// TIA Portal V16 export
// export: Created 2021-11-12T13:32:20.8858342Z, ExportSetting WithDefaults, DisplayName Totally Integrated Automation Portal, DisplayVersion V16 Update 3, DisplayName TIA Portal Version Control Interface, DisplayVersion V16 Update 2, DisplayName TIA Portal Openness, DisplayVersion V16 Update 3, DisplayName SINAMICS Startdrive Advanced, DisplayVersion V16 Update 5, DisplayName SINAMICS Startdrive G130, G150, S120, S150, SINAMICS MV, S210, DisplayVersion V16 Update 5, DisplayName SINAMICS Startdrive G110M, G120, G120C, G120D, G120P, G115D, DisplayVersion V16 Update 5, DisplayName STEP 7 Professional, DisplayVersion V16 Update 3, DisplayName STEP 7 Safety, DisplayVersion V16, DisplayName WinCC UA Professional, DisplayVersion V16 Update 3
DATA_BLOCK "HMI_PARAM_1R5"   // DB91
{ S7_Optimized_Access := 'TRUE' }
VERSION : 0.1
// stored: AutoNumber true, DBAccessibleFromOPCUA true, IsOnlyStoredInLoadMemory false, IsRetainMemResEnabled false, IsWriteProtectedInAS false, MemoryReserve 100
   VAR
      xxxxx___BinarySensors___xxxxx : Byte;
      "CL01-BG01_4" { S7_SetPoint := 'True'} : "UDT_CH_DI_Parameter";   // Robot 1R5 Gripper on table 1
      "CL01-BG02_4" { S7_SetPoint := 'True'} : "UDT_CH_DI_Parameter";   // Robot 1R5 Gripper on table 2
      xxxxx___BinaryOthers___xxxxx : Byte;
      PwrOK : "UDT_CH_DI_Parameter";
      "100+UH13-SF05_12" { S7_SetPoint := 'True'} : "UDT_CH_DI_Parameter";   // Robot 1R5 immediate stop
      "000+UH10-SF27_12" { S7_SetPoint := 'True'} : "UDT_CH_DI_Parameter";   // Okamžitý stop Robot 1R5
      xxxxx___AnalogueSensors___xxxxx : Byte;
      xxxxx___Drives___xxxxx : Byte;
      RO01 : "UDT_RobotABB_Parameter";   // Robot
      RC01 : "UDT_DriveRobotABB_Parameter";   // Controller
      Gripper : "UDT_RobotGripper_Parameter";   // Gripper
      xxxxx___Others___xxxxx : Byte;
      xxxxx__Alarms___xxxxx : Byte;
      RO01_Timeout : "UDT_DI_Mon_Parameter";   // Robot job active for too long
      CL01_BG01 { S7_SetPoint := 'True'} : "UDT_DI_Mon_Parameter";   // gripper on upper table
      CL01_BG02 { S7_SetPoint := 'True'} : "UDT_DI_Mon_Parameter";   // gripper on lower table
      ES { S7_SetPoint := 'True'} : "UDT_DI_Mon_Parameter";   // E-stop
   END_VAR
BEGIN
   "CL01-BG01_4".Color0 := 16#6;
   "CL01-BG01_4".Color1 := 16#0;
   CL01_BG01.Func := 16#6;
END_DATA_BLOCK
